Staubli VAL3: JTP.pgx

program JTP()
begin
  //建立坐标系
  setFrame(pt1,pt2,pt3,frmaster)
  //数据转换
  for nmaster=0 to 313
    pdemo[nmaster]=jointToPoint(t2,frmaster,master:ptRoutingPath[nmaster])
  endFor
end
